FUNCTION_BLOCK TwoConCtlCentralClient (* Composite Function Block Type *)
  (* Standard: 61499-2 *)
  (* Version 0.2, 2003-12-05, JHC, Rockwell Automation, Renamed from NEWCOMPFB. *)
  (* Version 0.1, 2002-01-08, JHC, Rockwell Automation, Added DLY FB as example. *)
  (* Version 0.0, 2000-05-27, JHC, Rockwell Automation *)
  (* Compiler header: package fb.rt.cs725; *)
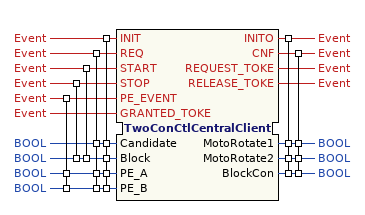
  EVENT_INPUT
    INIT WITH Candidate, Block, PE_A, PE_B; (* Initialization Request *)
    REQ WITH Candidate, PE_A, PE_B; (* Normal Execution Request *)
    START WITH Block;
    STOP WITH Block;
    PE_EVENT WITH PE_A, PE_B;
    GRANTED_TOKE;
  END_EVENT
  EVENT_OUTPUT
    INITO WITH MotoRotate1, MotoRotate2, BlockCon; (* Initialization Confirm *)
    CNF WITH MotoRotate1, MotoRotate2, BlockCon; (* Execution Confirmation *)
    REQUEST_TOKE;
    RELEASE_TOKE;
  END_EVENT
  VAR_INPUT
    Candidate : BOOL;
    Block : BOOL;
    PE_A : BOOL;
    PE_B : BOOL;
  END_VAR
  VAR_OUTPUT
    MotoRotate1 : BOOL;
    MotoRotate2 : BOOL;
    BlockCon : BOOL;
  END_VAR
  FBS
    FC11 : ConveyorCTL(Candidate := 0, Block := 0, PE := 0);
    Conv6Ctl : ConveyorCTLCentralClient;
  END_FBS
  EVENT_CONNECTIONS
    INIT TO FC11.INIT;
    REQ TO FC11.REQ;
    Conv6Ctl.INITO TO INITO;
    Conv6Ctl.CNF TO CNF;
    REQ TO Conv6Ctl.REQ;
    STOP TO Conv6Ctl.CAS_STOP;
    START TO Conv6Ctl.CAS_START;
    Conv6Ctl.STOP TO FC11.CAS_STOP;
    Conv6Ctl.START TO FC11.CAS_START;
    FC11.INITO TO Conv6Ctl.INIT;
    PE_EVENT TO Conv6Ctl.I_PE_EVENT;
    Conv6Ctl.REQUEST_TOKE TO REQUEST_TOKE;
    Conv6Ctl.RELEASE_TOKE TO RELEASE_TOKE;
    GRANTED_TOKE TO Conv6Ctl.GRANTED_TOKE;
  END_CONNECTIONS
  DATA_CONNECTIONS
    Block TO Conv6Ctl.Block;
    Candidate TO Conv6Ctl.Candidate;
    Conv6Ctl.BlockCon TO BlockCon;
    FC11.MotoRotate TO MotoRotate1;
    Conv6Ctl.MotoRotate TO MotoRotate2;
    PE_A TO Conv6Ctl.PE_IN;
    PE_B TO Conv6Ctl.PE_OUT;
  END_CONNECTIONS
END_FUNCTION_BLOCK
